TYPE T_PositiveDINT : DINT(0..2147483647); END_TYPE

(* stored: Version 1.1.0.1
   DUT T_PositiveDINT: Id {5fb6769a-9fa7-4d6c-8a4d-ea1ec6751abb} *)
